{attribute 'qualified_only'}
{attribute 'strict'}
{attribute 'to_string'}
TYPE DUT_Command_MoveType :
(
	CircularMove := 0,
	DirectMove := 1,
	LinearMove := 2
);
END_TYPE

(* stored: Version 1.1.0.1
   EnumerationTextList DUT_Command_MoveType: Id {6208825a-4125-41f0-8e7b-ec73206493b4} *)
